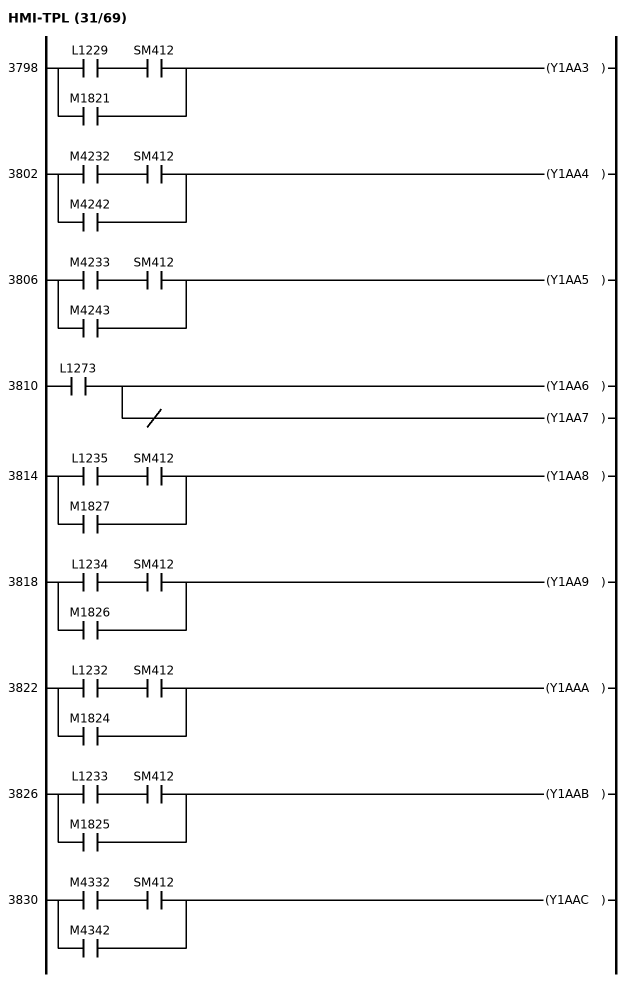
[picture p432: ladder of HMI-TPL, rungs at steps 3798 to 3830]
3798  LD      L1229
      AND     SM412
      OR      M1821
      OUT     Y1AA3
3802  LD      M4232
      AND     SM412
      OR      M4242
      OUT     Y1AA4
3806  LD      M4233
      AND     SM412
      OR      M4243
      OUT     Y1AA5
3810  LD      L1273
      OUT     Y1AA6
      INV
      OUT     Y1AA7
3814  LD      L1235
      AND     SM412
      OR      M1827
      OUT     Y1AA8
3818  LD      L1234
      AND     SM412
      OR      M1826
      OUT     Y1AA9
3822  LD      L1232
      AND     SM412
      OR      M1824
      OUT     Y1AAA
3826  LD      L1233
      AND     SM412
      OR      M1825
      OUT     Y1AAB
3830  LD      M4332
      AND     SM412
      OR      M4342
      OUT     Y1AAC
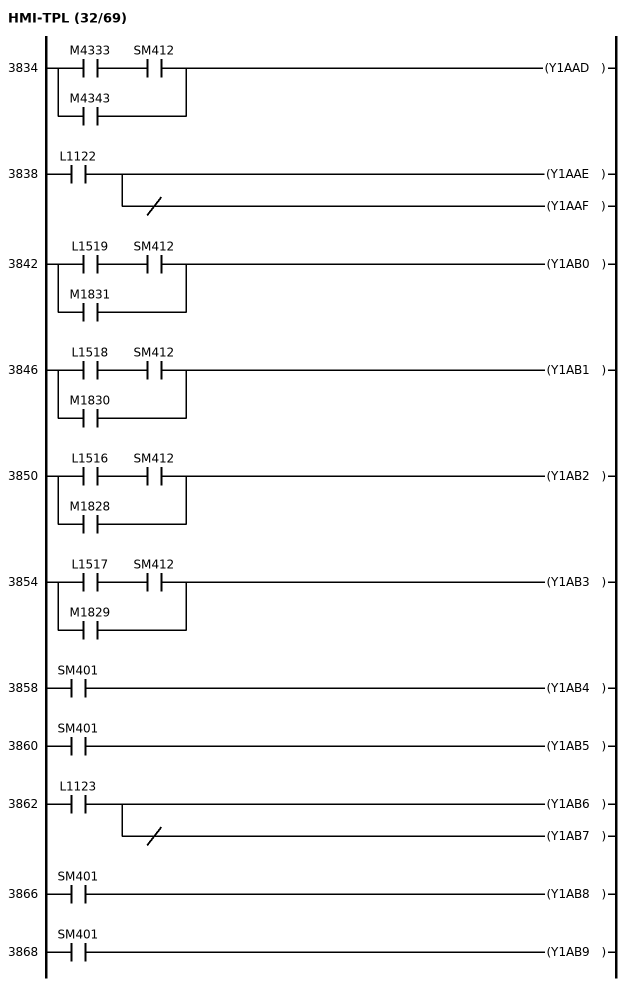
3834  LD      M4333
      AND     SM412
      OR      M4343
      OUT     Y1AAD
3838  LD      L1122
      OUT     Y1AAE
      INV
      OUT     Y1AAF
3842  LD      L1519
      AND     SM412
      OR      M1831
      OUT     Y1AB0
3846  LD      L1518
      AND     SM412
      OR      M1830
      OUT     Y1AB1
3850  LD      L1516
      AND     SM412
      OR      M1828
      OUT     Y1AB2
3854  LD      L1517
      AND     SM412
      OR      M1829
      OUT     Y1AB3
3858  LD      SM401
      OUT     Y1AB4
3860  LD      SM401
      OUT     Y1AB5
3862  LD      L1123
      OUT     Y1AB6
      INV
      OUT     Y1AB7
3866  LD      SM401
      OUT     Y1AB8
3868  LD      SM401
      OUT     Y1AB9
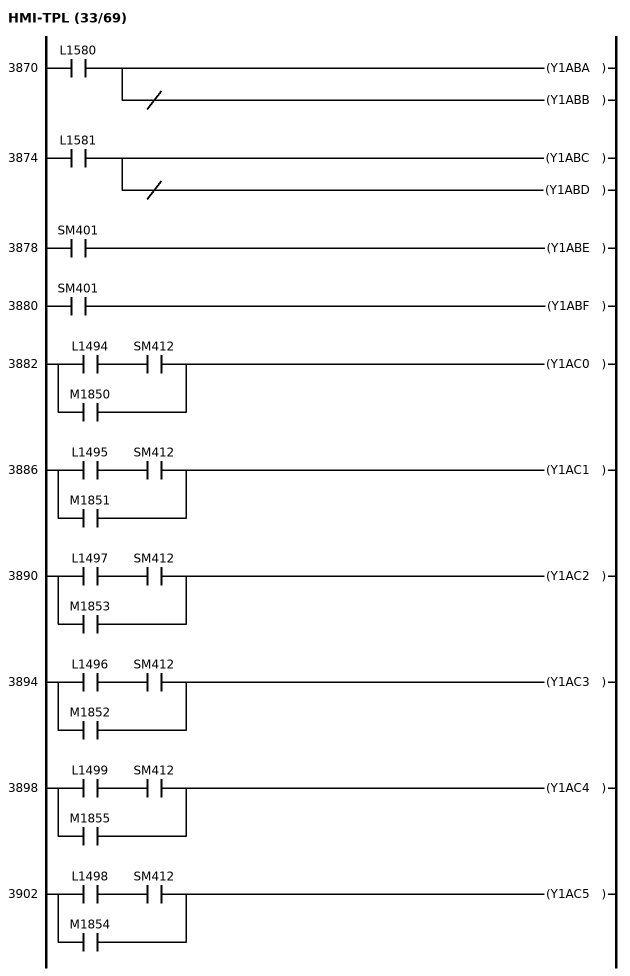
3870  LD      L1580
      OUT     Y1ABA
      INV
      OUT     Y1ABB
3874  LD      L1581
      OUT     Y1ABC
      INV
      OUT     Y1ABD
3878  LD      SM401
      OUT     Y1ABE
3880  LD      SM401
      OUT     Y1ABF
3882  LD      L1494
      AND     SM412
      OR      M1850
      OUT     Y1AC0
3886  LD      L1495
      AND     SM412
      OR      M1851
      OUT     Y1AC1
3890  LD      L1497
      AND     SM412
      OR      M1853
      OUT     Y1AC2
3894  LD      L1496
      AND     SM412
      OR      M1852
      OUT     Y1AC3
3898  LD      L1499
      AND     SM412
      OR      M1855
      OUT     Y1AC4
3902  LD      L1498
      AND     SM412
      OR      M1854
      OUT     Y1AC5
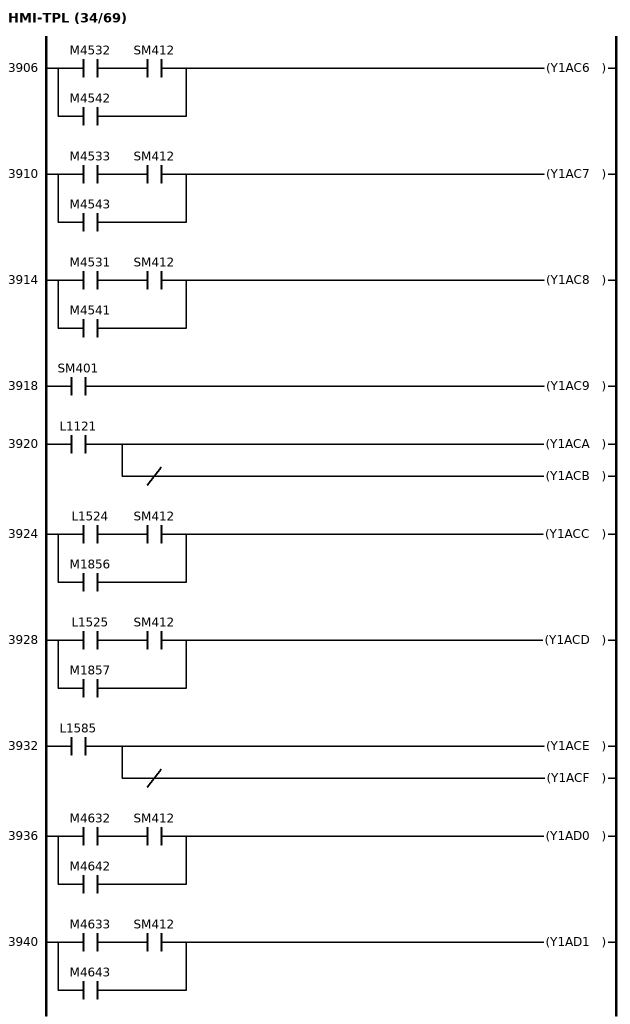
3906  LD      M4532
      AND     SM412
      OR      M4542
      OUT     Y1AC6
3910  LD      M4533
      AND     SM412
      OR      M4543
      OUT     Y1AC7
3914  LD      M4531
      AND     SM412
      OR      M4541
      OUT     Y1AC8
3918  LD      SM401
      OUT     Y1AC9
3920  LD      L1121
      OUT     Y1ACA
      INV
      OUT     Y1ACB
3924  LD      L1524
      AND     SM412
      OR      M1856
      OUT     Y1ACC
3928  LD      L1525
      AND     SM412
      OR      M1857
      OUT     Y1ACD
3932  LD      L1585
      OUT     Y1ACE
      INV
      OUT     Y1ACF
3936  LD      M4632
      AND     SM412
      OR      M4642
      OUT     Y1AD0
3940  LD      M4633
      AND     SM412
      OR      M4643
      OUT     Y1AD1
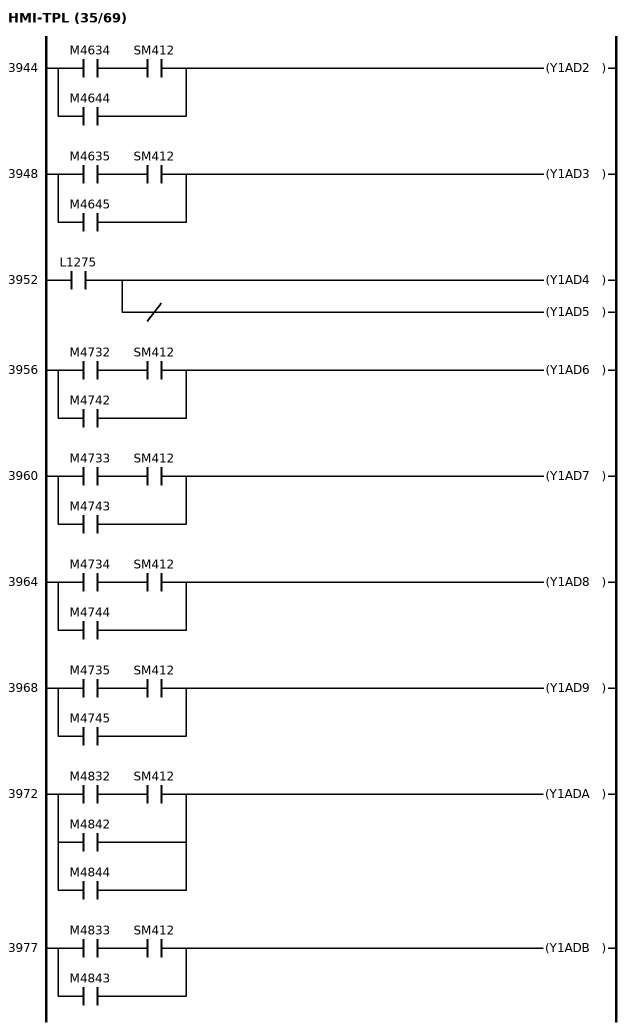
3944  LD      M4634
      AND     SM412
      OR      M4644
      OUT     Y1AD2
3948  LD      M4635
      AND     SM412
      OR      M4645
      OUT     Y1AD3
3952  LD      L1275
      OUT     Y1AD4
      INV
      OUT     Y1AD5
3956  LD      M4732
      AND     SM412
      OR      M4742
      OUT     Y1AD6
3960  LD      M4733
      AND     SM412
      OR      M4743
      OUT     Y1AD7
3964  LD      M4734
      AND     SM412
      OR      M4744
      OUT     Y1AD8
3968  LD      M4735
      AND     SM412
      OR      M4745
      OUT     Y1AD9
3972  LD      M4832
      AND     SM412
      OR      M4842
      OR      M4844
      OUT     Y1ADA
3977  LD      M4833
      AND     SM412
      OR      M4843
      OUT     Y1ADB
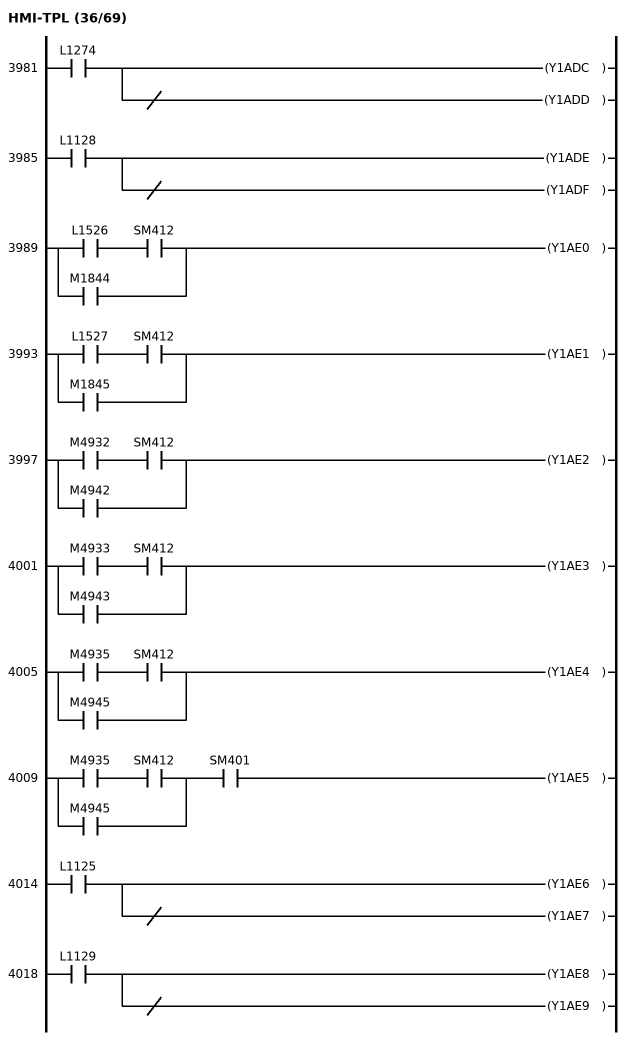
3981  LD      L1274
      OUT     Y1ADC
      INV
      OUT     Y1ADD
3985  LD      L1128
      OUT     Y1ADE
      INV
      OUT     Y1ADF
3989  LD      L1526
      AND     SM412
      OR      M1844
      OUT     Y1AE0
3993  LD      L1527
      AND     SM412
      OR      M1845
      OUT     Y1AE1
3997  LD      M4932
      AND     SM412
      OR      M4942
      OUT     Y1AE2
4001  LD      M4933
      AND     SM412
      OR      M4943
      OUT     Y1AE3
4005  LD      M4935
      AND     SM412
      OR      M4945
      OUT     Y1AE4
4009  LD      M4935
      AND     SM412
      OR      M4945
      AND     SM401
      OUT     Y1AE5
4014  LD      L1125
      OUT     Y1AE6
      INV
      OUT     Y1AE7
4018  LD      L1129
      OUT     Y1AE8
      INV
      OUT     Y1AE9
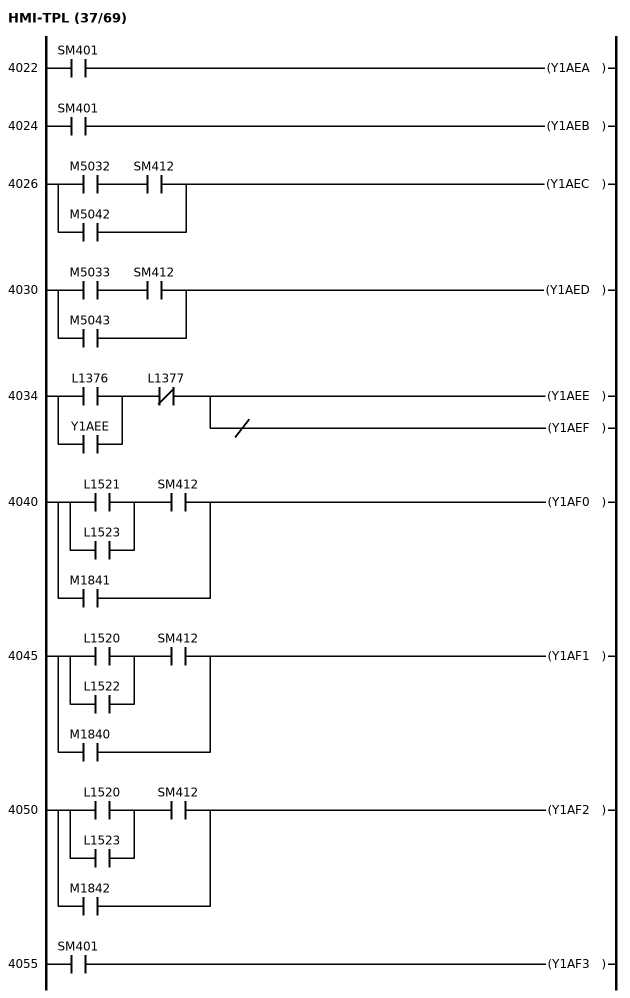
4022  LD      SM401
      OUT     Y1AEA
4024  LD      SM401
      OUT     Y1AEB
4026  LD      M5032
      AND     SM412
      OR      M5042
      OUT     Y1AEC
4030  LD      M5033
      AND     SM412
      OR      M5043
      OUT     Y1AED
4034  LD      L1376
      OR      Y1AEE
      ANI     L1377
      OUT     Y1AEE
      INV
      OUT     Y1AEF
4040  LD      L1521
      OR      L1523
      AND     SM412
      OR      M1841
      OUT     Y1AF0
4045  LD      L1520
      OR      L1522
      AND     SM412
      OR      M1840
      OUT     Y1AF1
4050  LD      L1520
      OR      L1523
      AND     SM412
      OR      M1842
      OUT     Y1AF2
4055  LD      SM401
      OUT     Y1AF3
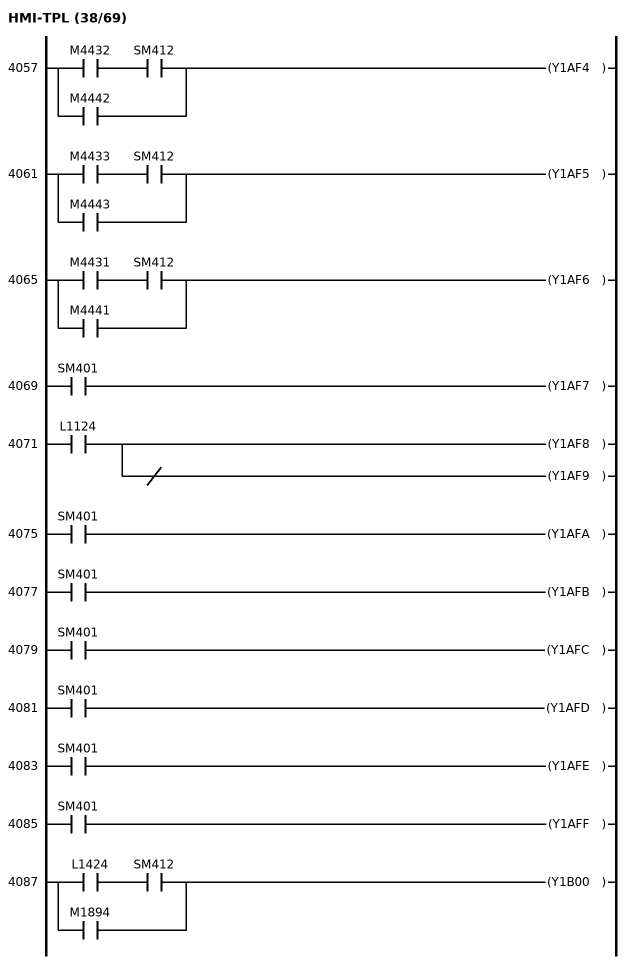
4057  LD      M4432
      AND     SM412
      OR      M4442
      OUT     Y1AF4
4061  LD      M4433
      AND     SM412
      OR      M4443
      OUT     Y1AF5
4065  LD      M4431
      AND     SM412
      OR      M4441
      OUT     Y1AF6
4069  LD      SM401
      OUT     Y1AF7
4071  LD      L1124
      OUT     Y1AF8
      INV
      OUT     Y1AF9
4075  LD      SM401
      OUT     Y1AFA
4077  LD      SM401
      OUT     Y1AFB
4079  LD      SM401
      OUT     Y1AFC
4081  LD      SM401
      OUT     Y1AFD
4083  LD      SM401
      OUT     Y1AFE
4085  LD      SM401
      OUT     Y1AFF
4087  LD      L1424
      AND     SM412
      OR      M1894
      OUT     Y1B00
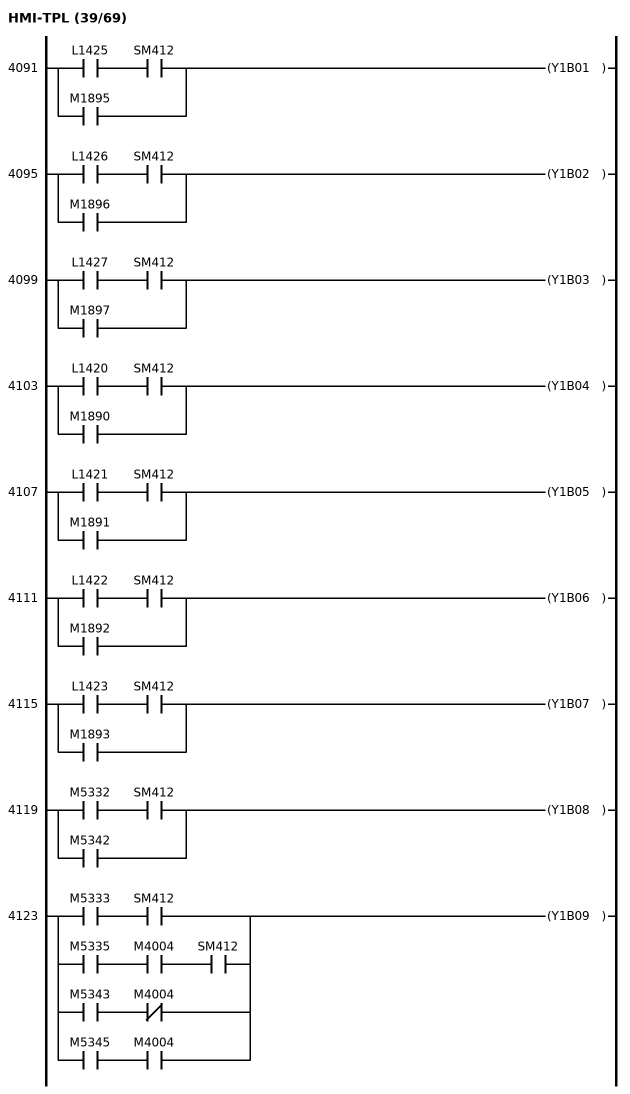
4091  LD      L1425
      AND     SM412
      OR      M1895
      OUT     Y1B01
4095  LD      L1426
      AND     SM412
      OR      M1896
      OUT     Y1B02
4099  LD      L1427
      AND     SM412
      OR      M1897
      OUT     Y1B03
4103  LD      L1420
      AND     SM412
      OR      M1890
      OUT     Y1B04
4107  LD      L1421
      AND     SM412
      OR      M1891
      OUT     Y1B05
4111  LD      L1422
      AND     SM412
      OR      M1892
      OUT     Y1B06
4115  LD      L1423
      AND     SM412
      OR      M1893
      OUT     Y1B07
4119  LD      M5332
      AND     SM412
      OR      M5342
      OUT     Y1B08
4123  LD      M5333
      AND     SM412
      LD      M5335
      AND     M4004
      AND     SM412
      ORB
      LD      M5343
      ANI     M4004
      ORB
      LD      M5345
      AND     M4004
      ORB
      OUT     Y1B09
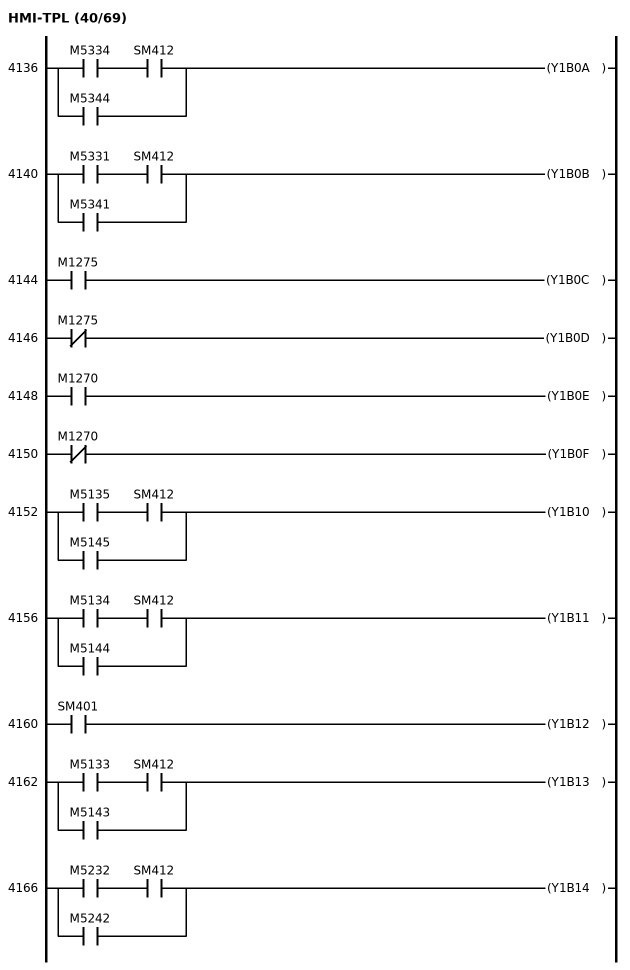
4136  LD      M5334
      AND     SM412
      OR      M5344
      OUT     Y1B0A
4140  LD      M5331
      AND     SM412
      OR      M5341
      OUT     Y1B0B
4144  LD      M1275
      OUT     Y1B0C
4146  LDI     M1275
      OUT     Y1B0D
4148  LD      M1270
      OUT     Y1B0E
4150  LDI     M1270
      OUT     Y1B0F
4152  LD      M5135
      AND     SM412
      OR      M5145
      OUT     Y1B10
4156  LD      M5134
      AND     SM412
      OR      M5144
      OUT     Y1B11
4160  LD      SM401
      OUT     Y1B12
4162  LD      M5133
      AND     SM412
      OR      M5143
      OUT     Y1B13
4166  LD      M5232
      AND     SM412
      OR      M5242
      OUT     Y1B14
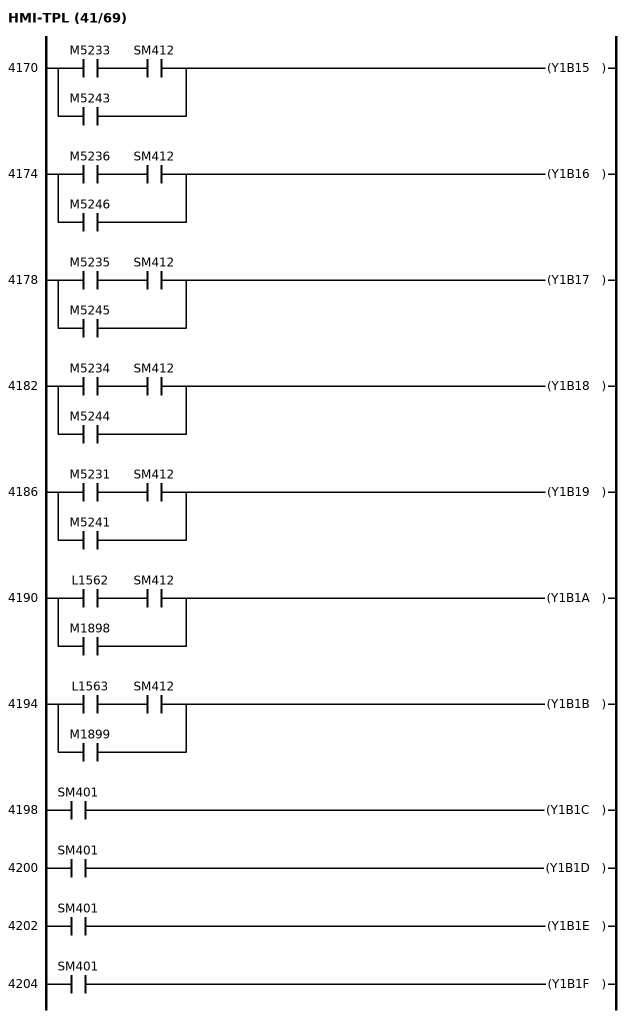
4170  LD      M5233
      AND     SM412
      OR      M5243
      OUT     Y1B15
4174  LD      M5236
      AND     SM412
      OR      M5246
      OUT     Y1B16
4178  LD      M5235
      AND     SM412
      OR      M5245
      OUT     Y1B17
4182  LD      M5234
      AND     SM412
      OR      M5244
      OUT     Y1B18
4186  LD      M5231
      AND     SM412
      OR      M5241
      OUT     Y1B19
4190  LD      L1562
      AND     SM412
      OR      M1898
      OUT     Y1B1A
4194  LD      L1563
      AND     SM412
      OR      M1899
      OUT     Y1B1B
4198  LD      SM401
      OUT     Y1B1C
4200  LD      SM401
      OUT     Y1B1D
4202  LD      SM401
      OUT     Y1B1E
4204  LD      SM401
      OUT     Y1B1F
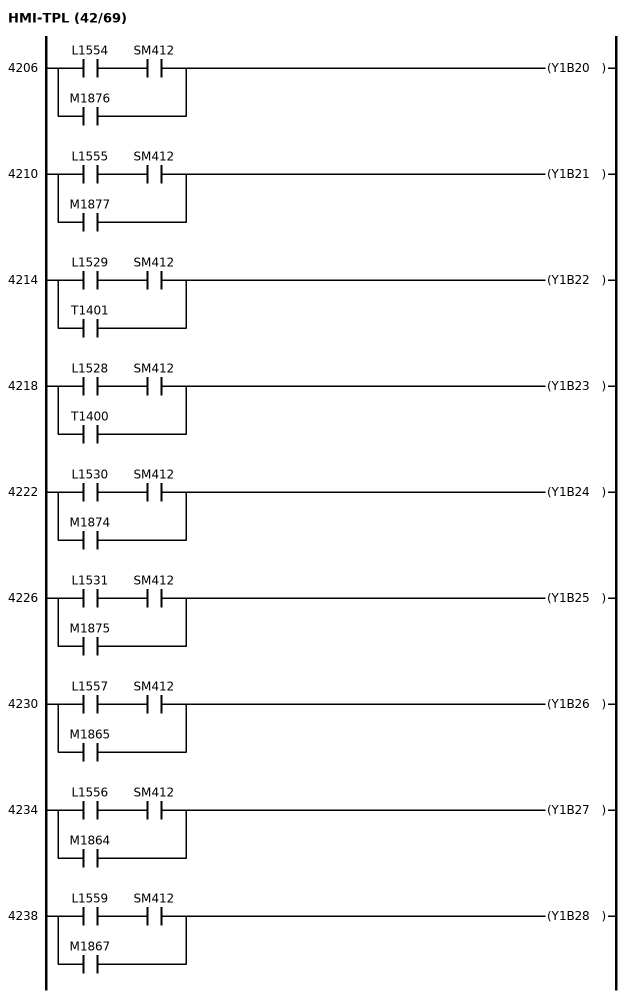
4206  LD      L1554
      AND     SM412
      OR      M1876
      OUT     Y1B20
4210  LD      L1555
      AND     SM412
      OR      M1877
      OUT     Y1B21
4214  LD      L1529
      AND     SM412
      OR      T1401
      OUT     Y1B22
4218  LD      L1528
      AND     SM412
      OR      T1400
      OUT     Y1B23
4222  LD      L1530
      AND     SM412
      OR      M1874
      OUT     Y1B24
4226  LD      L1531
      AND     SM412
      OR      M1875
      OUT     Y1B25
4230  LD      L1557
      AND     SM412
      OR      M1865
      OUT     Y1B26
4234  LD      L1556
      AND     SM412
      OR      M1864
      OUT     Y1B27
4238  LD      L1559
      AND     SM412
      OR      M1867
      OUT     Y1B28
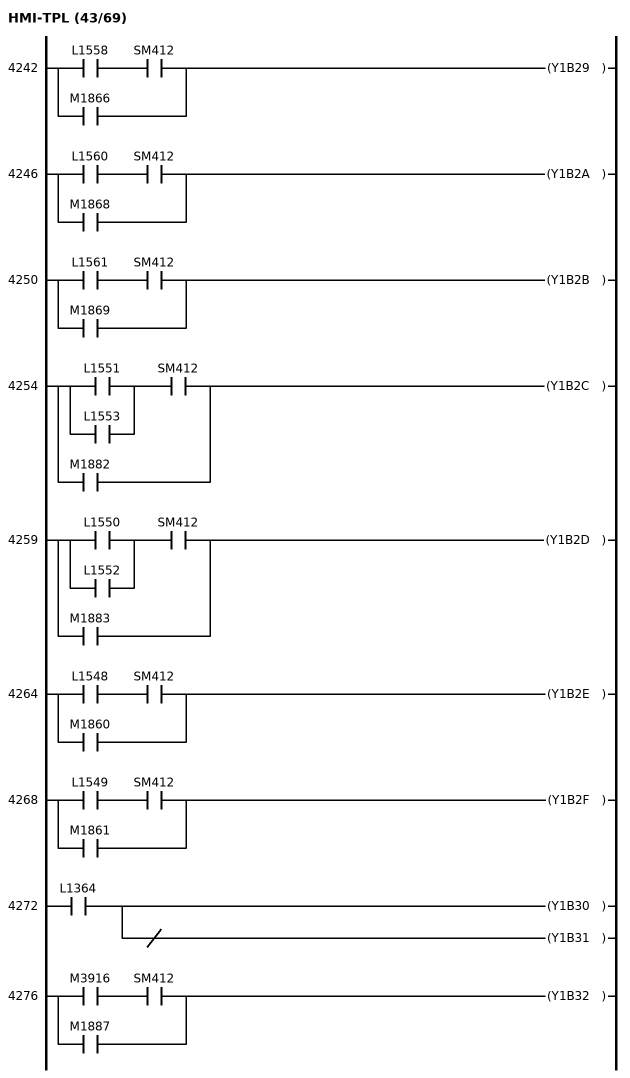
4242  LD      L1558
      AND     SM412
      OR      M1866
      OUT     Y1B29
4246  LD      L1560
      AND     SM412
      OR      M1868
      OUT     Y1B2A
4250  LD      L1561
      AND     SM412
      OR      M1869
      OUT     Y1B2B
4254  LD      L1551
      OR      L1553
      AND     SM412
      OR      M1882
      OUT     Y1B2C
4259  LD      L1550
      OR      L1552
      AND     SM412
      OR      M1883
      OUT     Y1B2D
4264  LD      L1548
      AND     SM412
      OR      M1860
      OUT     Y1B2E
4268  LD      L1549
      AND     SM412
      OR      M1861
      OUT     Y1B2F
4272  LD      L1364
      OUT     Y1B30
      INV
      OUT     Y1B31
4276  LD      M3916
      AND     SM412
      OR      M1887
      OUT     Y1B32
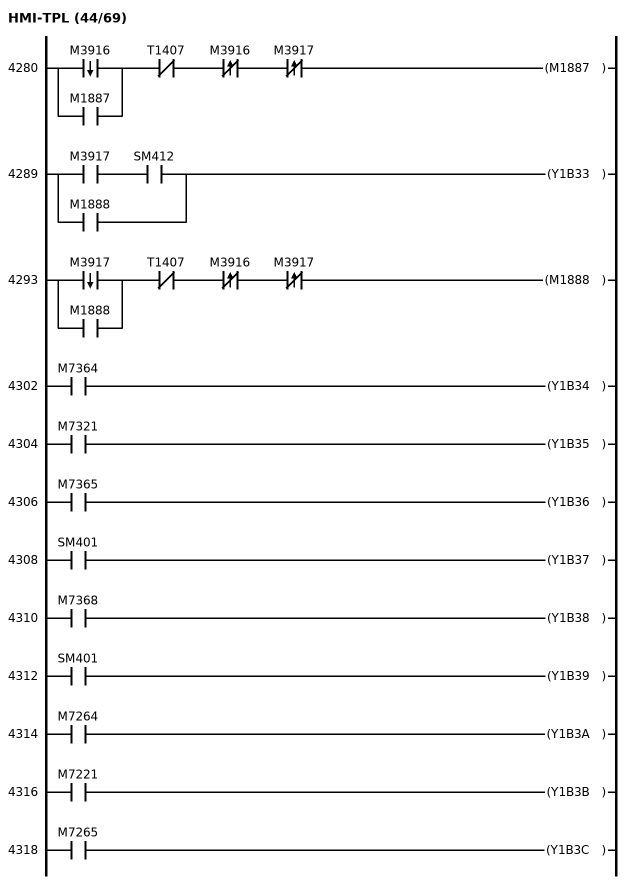
4280  LDF     M3916
      OR      M1887
      ANI     T1407
      ANDPI   M3916
      ANDPI   M3917
      OUT     M1887
4289  LD      M3917
      AND     SM412
      OR      M1888
      OUT     Y1B33
4293  LDF     M3917
      OR      M1888
      ANI     T1407
      ANDPI   M3916
      ANDPI   M3917
      OUT     M1888
4302  LD      M7364
      OUT     Y1B34
4304  LD      M7321
      OUT     Y1B35
4306  LD      M7365
      OUT     Y1B36
4308  LD      SM401
      OUT     Y1B37
4310  LD      M7368
      OUT     Y1B38
4312  LD      SM401
      OUT     Y1B39
4314  LD      M7264
      OUT     Y1B3A
4316  LD      M7221
      OUT     Y1B3B
4318  LD      M7265
      OUT     Y1B3C
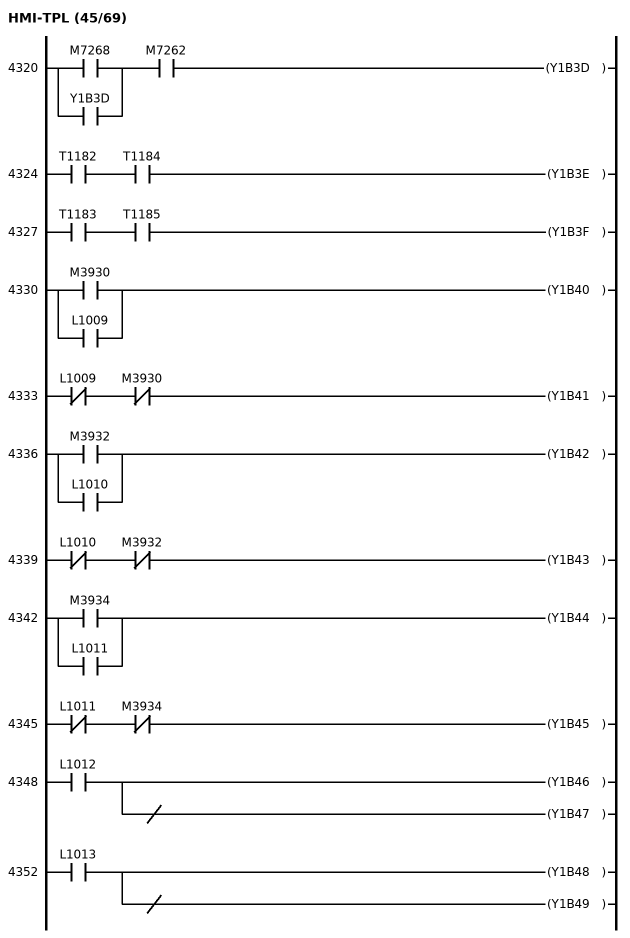
4320  LD      M7268
      OR      Y1B3D
      AND     M7262
      OUT     Y1B3D
4324  LD      T1182
      AND     T1184
      OUT     Y1B3E
4327  LD      T1183
      AND     T1185
      OUT     Y1B3F
4330  LD      M3930
      OR      L1009
      OUT     Y1B40
4333  LDI     L1009
      ANI     M3930
      OUT     Y1B41
4336  LD      M3932
      OR      L1010
      OUT     Y1B42
4339  LDI     L1010
      ANI     M3932
      OUT     Y1B43
4342  LD      M3934
      OR      L1011
      OUT     Y1B44
4345  LDI     L1011
      ANI     M3934
      OUT     Y1B45
4348  LD      L1012
      OUT     Y1B46
      INV
      OUT     Y1B47
4352  LD      L1013
      OUT     Y1B48
      INV
      OUT     Y1B49
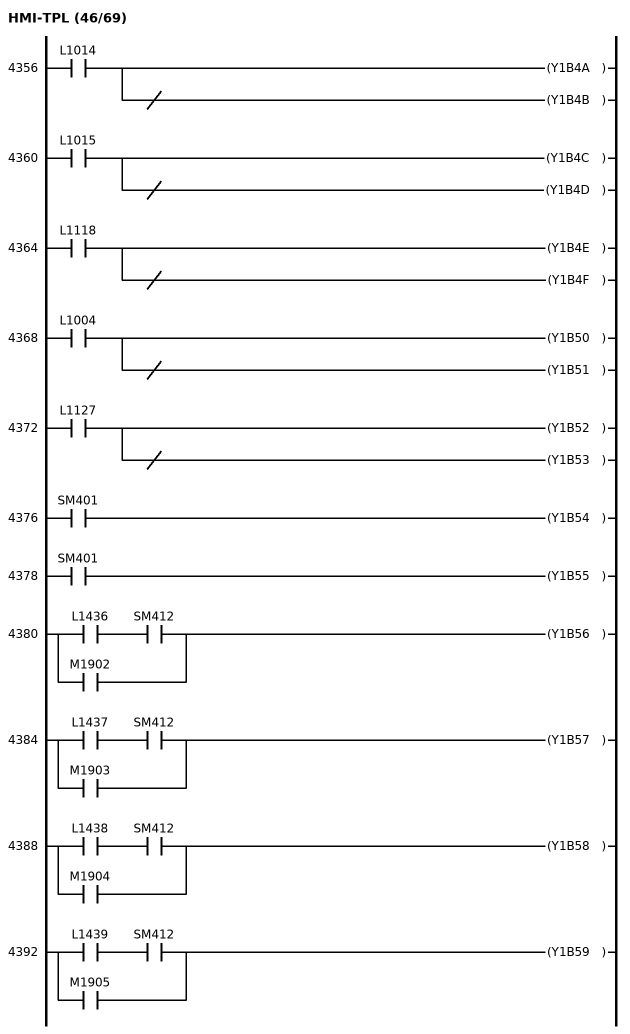
4356  LD      L1014
      OUT     Y1B4A
      INV
      OUT     Y1B4B
4360  LD      L1015
      OUT     Y1B4C
      INV
      OUT     Y1B4D
4364  LD      L1118
      OUT     Y1B4E
      INV
      OUT     Y1B4F
4368  LD      L1004
      OUT     Y1B50
      INV
      OUT     Y1B51
4372  LD      L1127
      OUT     Y1B52
      INV
      OUT     Y1B53
4376  LD      SM401
      OUT     Y1B54
4378  LD      SM401
      OUT     Y1B55
4380  LD      L1436
      AND     SM412
      OR      M1902
      OUT     Y1B56
4384  LD      L1437
      AND     SM412
      OR      M1903
      OUT     Y1B57
4388  LD      L1438
      AND     SM412
      OR      M1904
      OUT     Y1B58
4392  LD      L1439
      AND     SM412
      OR      M1905
      OUT     Y1B59
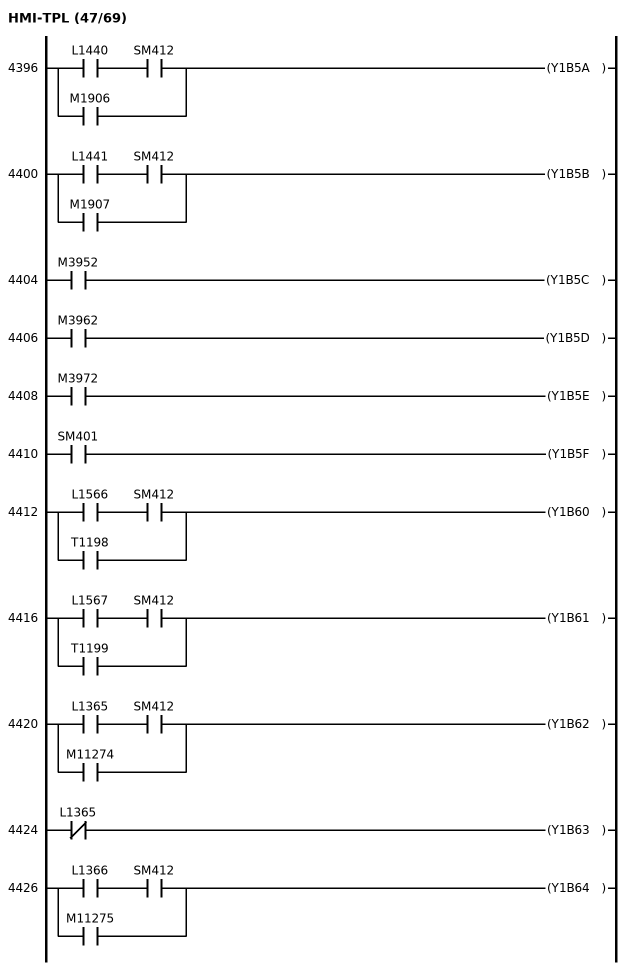
4396  LD      L1440
      AND     SM412
      OR      M1906
      OUT     Y1B5A
4400  LD      L1441
      AND     SM412
      OR      M1907
      OUT     Y1B5B
4404  LD      M3952
      OUT     Y1B5C
4406  LD      M3962
      OUT     Y1B5D
4408  LD      M3972
      OUT     Y1B5E
4410  LD      SM401
      OUT     Y1B5F
4412  LD      L1566
      AND     SM412
      OR      T1198
      OUT     Y1B60
4416  LD      L1567
      AND     SM412
      OR      T1199
      OUT     Y1B61
4420  LD      L1365
      AND     SM412
      OR      M11274
      OUT     Y1B62
4424  LDI     L1365
      OUT     Y1B63
4426  LD      L1366
      AND     SM412
      OR      M11275
      OUT     Y1B64
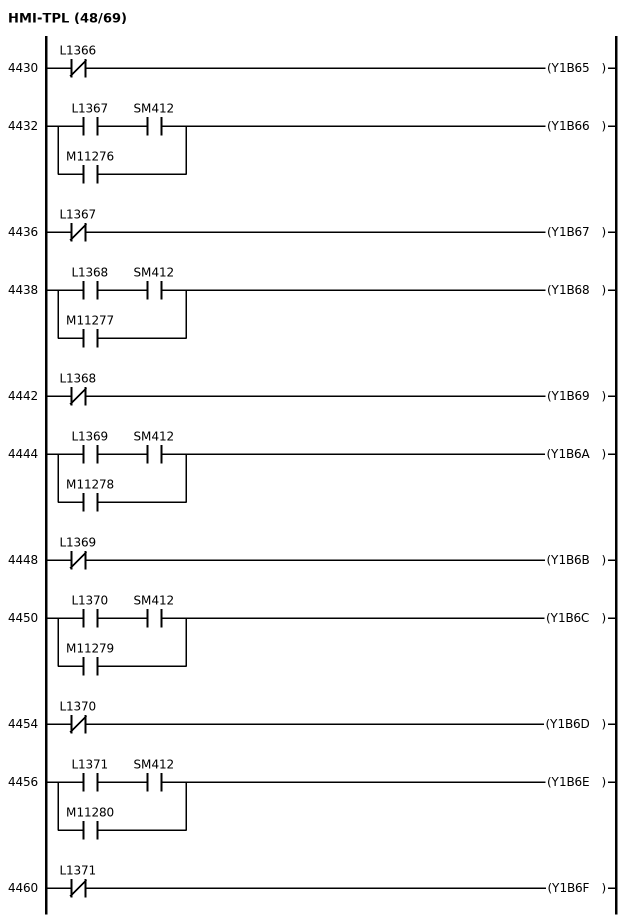
4430  LDI     L1366
      OUT     Y1B65
4432  LD      L1367
      AND     SM412
      OR      M11276
      OUT     Y1B66
4436  LDI     L1367
      OUT     Y1B67
4438  LD      L1368
      AND     SM412
      OR      M11277
      OUT     Y1B68
4442  LDI     L1368
      OUT     Y1B69
4444  LD      L1369
      AND     SM412
      OR      M11278
      OUT     Y1B6A
4448  LDI     L1369
      OUT     Y1B6B
4450  LD      L1370
      AND     SM412
      OR      M11279
      OUT     Y1B6C
4454  LDI     L1370
      OUT     Y1B6D
4456  LD      L1371
      AND     SM412
      OR      M11280
      OUT     Y1B6E
4460  LDI     L1371
      OUT     Y1B6F
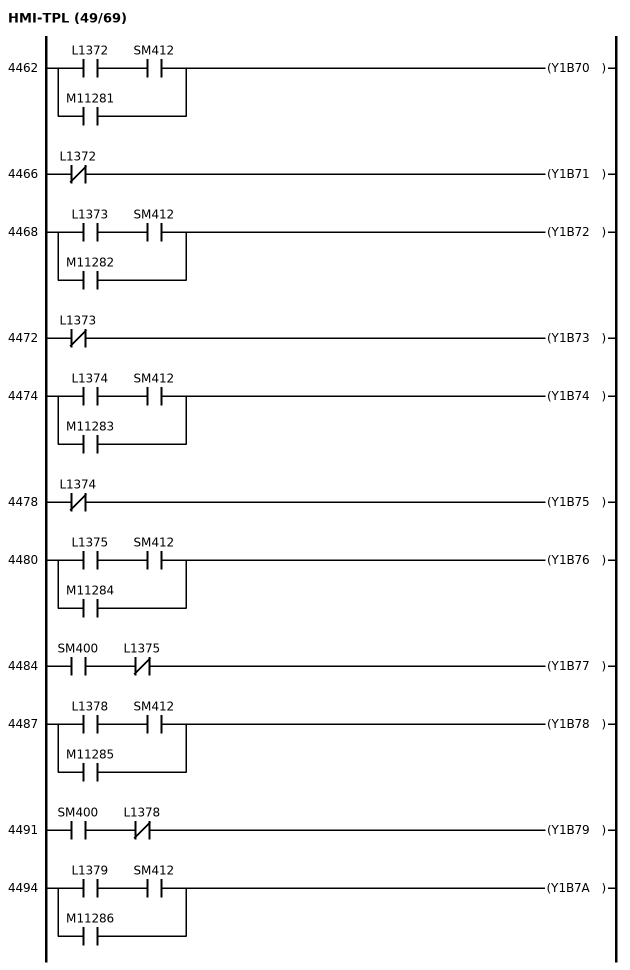
4462  LD      L1372
      AND     SM412
      OR      M11281
      OUT     Y1B70
4466  LDI     L1372
      OUT     Y1B71
4468  LD      L1373
      AND     SM412
      OR      M11282
      OUT     Y1B72
4472  LDI     L1373
      OUT     Y1B73
4474  LD      L1374
      AND     SM412
      OR      M11283
      OUT     Y1B74
4478  LDI     L1374
      OUT     Y1B75
4480  LD      L1375
      AND     SM412
      OR      M11284
      OUT     Y1B76
4484  LD      SM400
      ANI     L1375
      OUT     Y1B77
4487  LD      L1378
      AND     SM412
      OR      M11285
      OUT     Y1B78
4491  LD      SM400
      ANI     L1378
      OUT     Y1B79
4494  LD      L1379
      AND     SM412
      OR      M11286
      OUT     Y1B7A
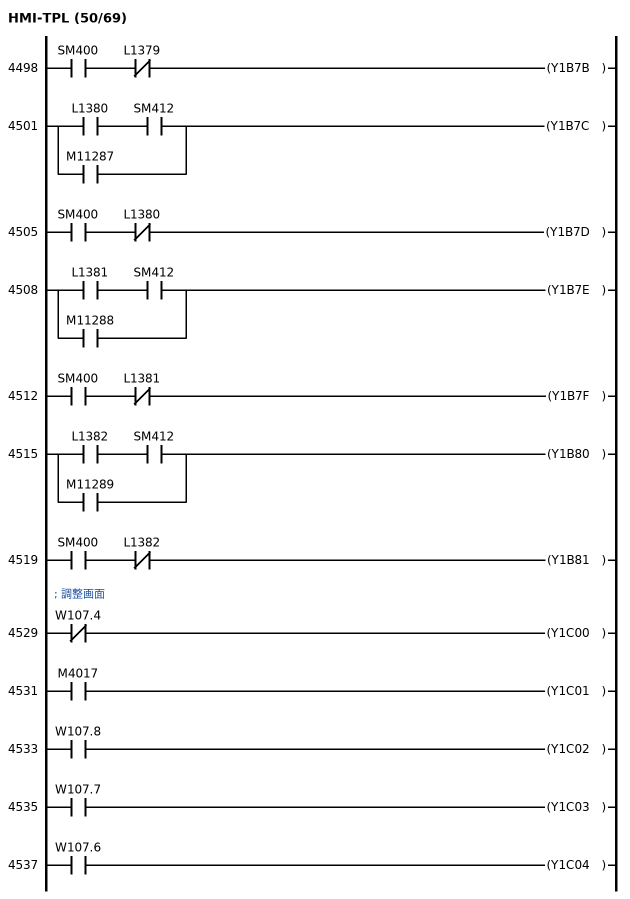
4498  LD      SM400
      ANI     L1379
      OUT     Y1B7B
4501  LD      L1380
      AND     SM412
      OR      M11287
      OUT     Y1B7C
4505  LD      SM400
      ANI     L1380
      OUT     Y1B7D
4508  LD      L1381
      AND     SM412
      OR      M11288
      OUT     Y1B7E
4512  LD      SM400
      ANI     L1381
      OUT     Y1B7F
4515  LD      L1382
      AND     SM412
      OR      M11289
      OUT     Y1B80
4519  LD      SM400
      ANI     L1382
      OUT     Y1B81
; 調整画面
4529  LDI     W107.4
      OUT     Y1C00
4531  LD      M4017
      OUT     Y1C01
4533  LD      W107.8
      OUT     Y1C02
4535  LD      W107.7
      OUT     Y1C03
4537  LD      W107.6
      OUT     Y1C04
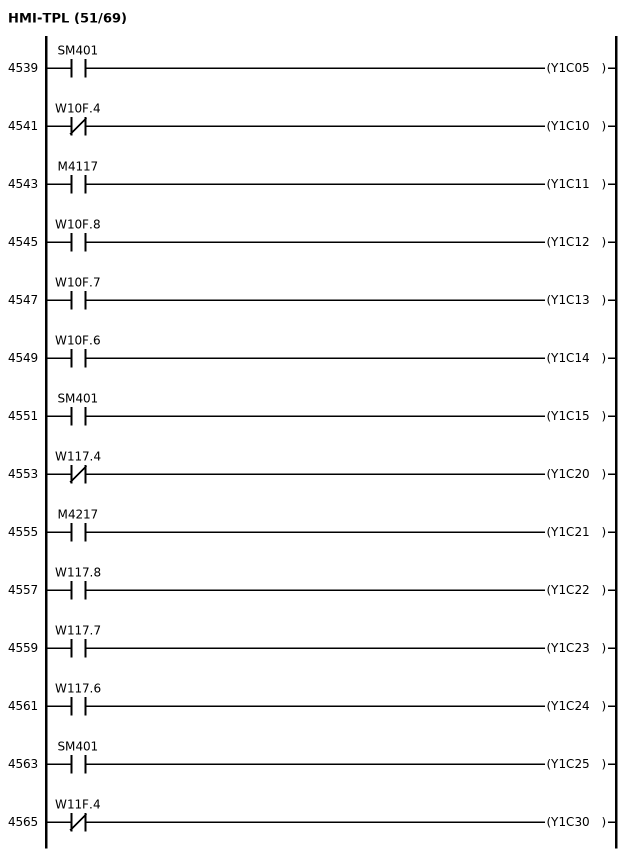
4539  LD      SM401
      OUT     Y1C05
4541  LDI     W10F.4
      OUT     Y1C10
4543  LD      M4117
      OUT     Y1C11
4545  LD      W10F.8
      OUT     Y1C12
4547  LD      W10F.7
      OUT     Y1C13
4549  LD      W10F.6
      OUT     Y1C14
4551  LD      SM401
      OUT     Y1C15
4553  LDI     W117.4
      OUT     Y1C20
4555  LD      M4217
      OUT     Y1C21
4557  LD      W117.8
      OUT     Y1C22
4559  LD      W117.7
      OUT     Y1C23
4561  LD      W117.6
      OUT     Y1C24
4563  LD      SM401
      OUT     Y1C25
4565  LDI     W11F.4
      OUT     Y1C30
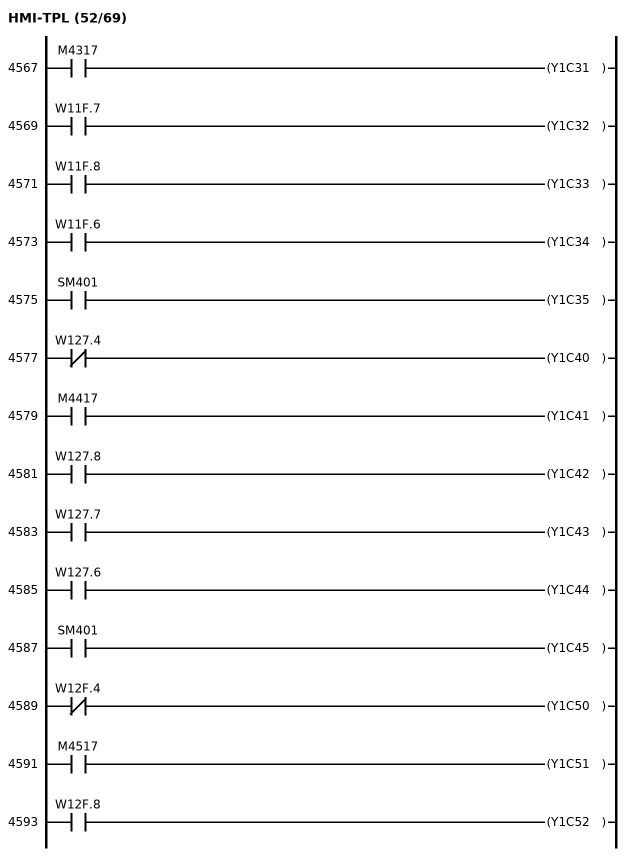
4567  LD      M4317
      OUT     Y1C31
4569  LD      W11F.7
      OUT     Y1C32
4571  LD      W11F.8
      OUT     Y1C33
4573  LD      W11F.6
      OUT     Y1C34
4575  LD      SM401
      OUT     Y1C35
4577  LDI     W127.4
      OUT     Y1C40
4579  LD      M4417
      OUT     Y1C41
4581  LD      W127.8
      OUT     Y1C42
4583  LD      W127.7
      OUT     Y1C43
4585  LD      W127.6
      OUT     Y1C44
4587  LD      SM401
      OUT     Y1C45
4589  LDI     W12F.4
      OUT     Y1C50
4591  LD      M4517
      OUT     Y1C51
4593  LD      W12F.8
      OUT     Y1C52
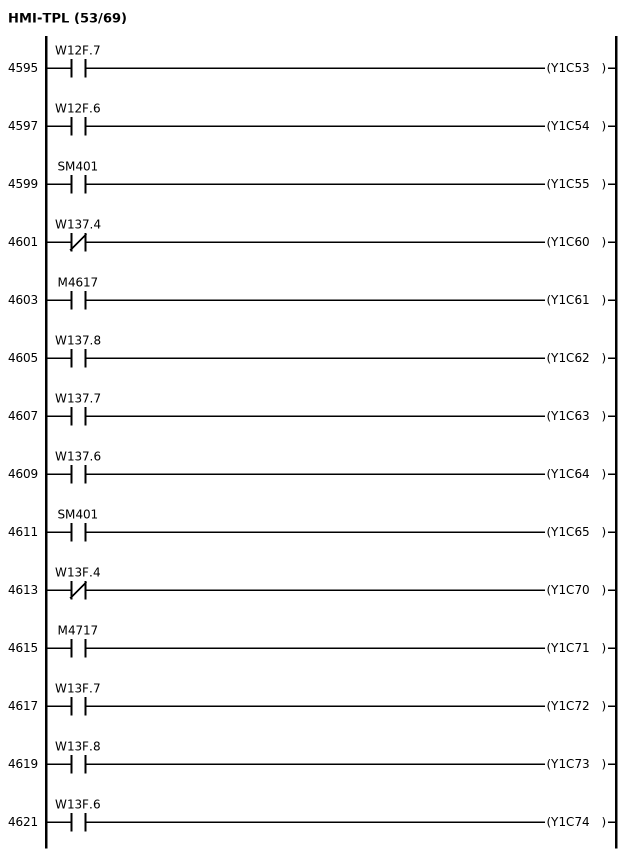
4595  LD      W12F.7
      OUT     Y1C53
4597  LD      W12F.6
      OUT     Y1C54
4599  LD      SM401
      OUT     Y1C55
4601  LDI     W137.4
      OUT     Y1C60
4603  LD      M4617
      OUT     Y1C61
4605  LD      W137.8
      OUT     Y1C62
4607  LD      W137.7
      OUT     Y1C63
4609  LD      W137.6
      OUT     Y1C64
4611  LD      SM401
      OUT     Y1C65
4613  LDI     W13F.4
      OUT     Y1C70
4615  LD      M4717
      OUT     Y1C71
4617  LD      W13F.7
      OUT     Y1C72
4619  LD      W13F.8
      OUT     Y1C73
4621  LD      W13F.6
      OUT     Y1C74
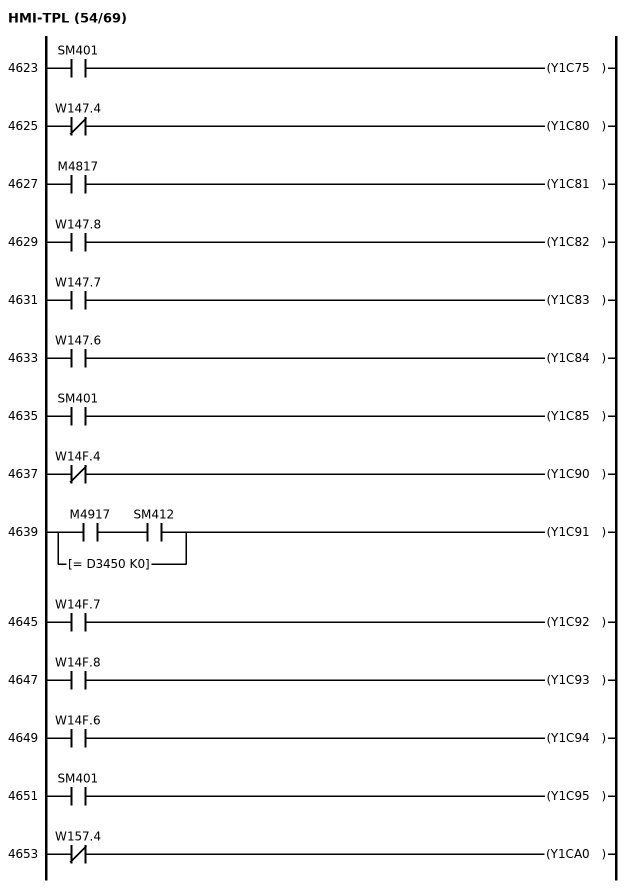
4623  LD      SM401
      OUT     Y1C75
4625  LDI     W147.4
      OUT     Y1C80
4627  LD      M4817
      OUT     Y1C81
4629  LD      W147.8
      OUT     Y1C82
4631  LD      W147.7
      OUT     Y1C83
4633  LD      W147.6
      OUT     Y1C84
4635  LD      SM401
      OUT     Y1C85
4637  LDI     W14F.4
      OUT     Y1C90
4639  LD      M4917
      AND     SM412
      OR=     D3450 K0
      OUT     Y1C91
4645  LD      W14F.7
      OUT     Y1C92
4647  LD      W14F.8
      OUT     Y1C93
4649  LD      W14F.6
      OUT     Y1C94
4651  LD      SM401
      OUT     Y1C95
4653  LDI     W157.4
      OUT     Y1CA0
